TEXTLIST DUT_types
  0 = 'Etalon 1'
  1 = 'Etalon 2'
  2 = 'Etalon 3'
  3 = 'Termék'
   = ''
END_TEXTLIST

(* stored: Version 1.1.0.1, ProductVersion 3.1.4020.3
   TextList DUT_types: Id {f228ab42-086d-4dd6-8346-7c81ee115dfd} *)
